ABB RAPID module: SetupWO.mod

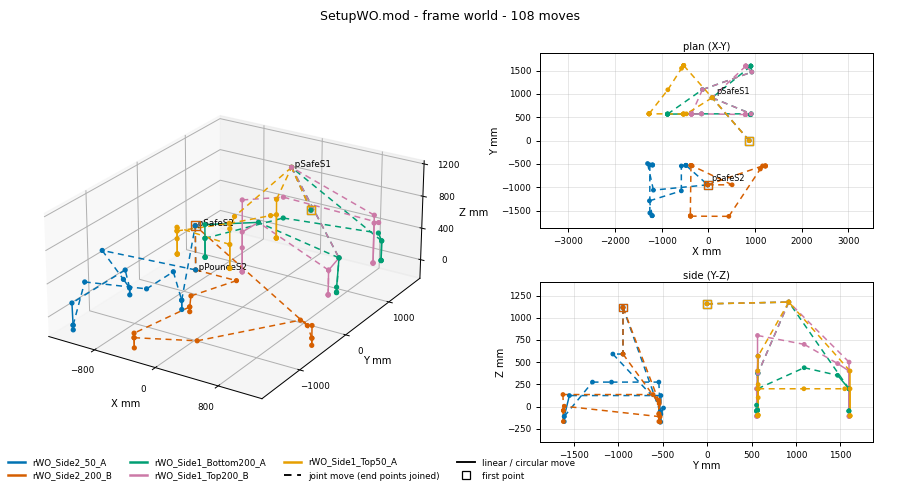
[picture p0: tool path of SetupWO.mod in frame world, 108 of 108 moves have a stored position in this frame; points joined in program order, loops and branches not executed]
MODULE SetupWO
	CONST robtarget pPounceS11:=[[-35.68,-1481.68,-160.88],[0.0139857,0.369962,0.928841,-0.0136566],[-2,1,-2,0],[9E+09,9E+09,9E+09,9E+09,9E+09,9E+09]];
	CONST robtarget pPounceS12:=[[1323.92,1454.10,-169.98],[0.00216079,-0.276188,0.961084,0.00568097],[0,-2,1,0],[9E+09,9E+09,9E+09,9E+09,9E+09,9E+09]];
	CONST robtarget pSafeS91:=[[-851.55,865.08,638.38],[0.0987927,0.977932,-0.183201,0.0180468],[1,0,-1,0],[9E+09,9E+09,9E+09,9E+09,9E+09,9E+09]];
	PROC rWO_Side2_50_A()
		MoveJ pSafeS2, v800, fine, tWeldGun;
		MoveJ pPounceS2, v800, fine, tWeldGun;
		MoveJ [[-1175.59,-1061.41,590.91],[0.0290518,0.998376,-0.0425584,0.0242723],[-2,-1,0,0],[9E+09,9E+09,9E+09,9E+09,9E+09,9E+09]], v800, z10, tWeldGun;
		MoveJ [[-1300.83,-491.42,-17.13],[0.0290285,0.998379,-0.0425044,0.0242811],[-2,-2,1,0],[9E+09,9E+09,9E+09,9E+09,9E+09,9E+09]], v800, z10, tWeldGun;
		MoveL [[-1195.07,-522.25,-85.28],[0.0287714,0.998373,-0.0426242,0.0246318],[-2,-2,1,0],[9E+09,9E+09,9E+09,9E+09,9E+09,9E+09]], v800, z10, tWeldGun;
		X1:
		MoveL [[-1195.09,-522.33,-173.98],[0.0287773,0.998376,-0.042547,0.0246393],[-2,-2,1,0],[9E+09,9E+09,9E+09,9E+09,9E+09,9E+09]], v800, fine, tWeldGun;
		MoveL [[-1195.07,-522.24,-85.28],[0.0287708,0.998373,-0.0426249,0.0246327],[-2,-2,1,0],[9E+09,9E+09,9E+09,9E+09,9E+09,9E+09]], v800, z10, tWeldGun;
		MoveJ [[-1253.08,-520.20,123.53],[0.0289856,0.998373,-0.0426291,0.0243837],[-2,-2,1,0],[9E+09,9E+09,9E+09,9E+09,9E+09,9E+09]], v800, z10, tWeldGun;
		MoveJ [[-1252.34,-1550.77,123.51],[0.0289915,0.998371,-0.0426611,0.0243853],[-2,-1,1,0],[9E+09,9E+09,9E+09,9E+09,9E+09,9E+09]], v800, z10, tWeldGun;
		MoveL [[-1203.52,-1608.74,-112.11],[0.0144898,0.998681,-0.0423691,0.0251074],[-2,-1,1,0],[9E+09,9E+09,9E+09,9E+09,9E+09,9E+09]], v800, z10, tWeldGun;
		X2:
		MoveL [[-1203.58,-1608.77,-169.27],[0.0144836,0.998684,-0.0423489,0.025044],[-2,-1,1,0],[9E+09,9E+09,9E+09,9E+09,9E+09,9E+09]], v800, fine, tWeldGun;
		MoveL [[-1203.52,-1608.74,-112.11],[0.0144918,0.998681,-0.0423701,0.0251105],[-2,-1,1,0],[9E+09,9E+09,9E+09,9E+09,9E+09,9E+09]], v800, z10, tWeldGun;
		MoveJ [[-1260.62,-1290.63,274.96],[0.0145241,0.998684,-0.0422942,0.0250997],[-2,-1,1,0],[9E+09,9E+09,9E+09,9E+09,9E+09,9E+09]], v800, z10, tWeldGun;
		MoveJ [[-577.42,-1076.50,274.99],[0.0145152,0.998684,-0.042322,0.0250813],[-2,-1,1,0],[9E+09,9E+09,9E+09,9E+09,9E+09,9E+09]], v800, z10, tWeldGun;
		MoveJ [[-577.39,-543.42,274.98],[0.0145354,0.998682,-0.0423423,0.0251146],[-2,-1,1,0],[9E+09,9E+09,9E+09,9E+09,9E+09,9E+09]], v800, z10, tWeldGun;
		MoveJ [[-478.99,-529.16,-59.08],[0.0144521,0.998675,-0.0425363,0.0251153],[-2,-2,1,0],[9E+09,9E+09,9E+09,9E+09,9E+09,9E+09]], v800, z10, tWeldGun;
		Y1:
		MoveL [[-479.00,-529.24,-174.87],[0.0144769,0.998677,-0.0424711,0.0251064],[-2,-2,2,0],[9E+09,9E+09,9E+09,9E+09,9E+09,9E+09]], v800, fine, tWeldGun;
		MoveL [[-478.99,-529.16,-59.08],[0.0144527,0.998675,-0.0425336,0.0251147],[-2,-2,1,0],[9E+09,9E+09,9E+09,9E+09,9E+09,9E+09]], v800, z10, tWeldGun;
		MoveJ pSafeS2, v800, fine, tWeldGun;
	ENDPROC
	PROC rWO_Side2_200_B()
		MoveJ pSafeS2, v800, fine, tWeldGun;
		MoveJ pPounceS2, v800, fine, tWeldGun;
		MoveJ [[510.39,-947.34,590.96],[0.00440116,-0.169072,0.985593,-0.00107979],[-1,0,-2,0],[9E+09,9E+09,9E+09,9E+09,9E+09,9E+09]], v800, z10, tWeldGun;
		MoveJ [[-346.53,-539.81,31.85],[0.00581128,-0.165183,0.98623,-0.00561328],[-2,0,-2,0],[9E+09,9E+09,9E+09,9E+09,9E+09,9E+09]], v800, z10, tWeldGun;
		MoveL [[-370.69,-531.16,-114.28],[0.00581574,-0.165115,0.986242,-0.00552901],[-2,0,-2,0],[9E+09,9E+09,9E+09,9E+09,9E+09,9E+09]], v800, z10, tWeldGun;
		X1:
		MoveL [[-370.69,-531.24,-173.68],[0.00581718,-0.165073,0.986249,-0.00556015],[-2,0,-2,0],[9E+09,9E+09,9E+09,9E+09,9E+09,9E+09]], v800, fine, tWeldGun;
		MoveL [[-370.69,-531.16,-114.28],[0.00581398,-0.165115,0.986242,-0.00552968],[-2,0,-2,0],[9E+09,9E+09,9E+09,9E+09,9E+09,9E+09]], v800, z10, tWeldGun;
		MoveJ [[-385.03,-1608.16,3.65],[0.0114791,0.162686,-0.986611,-0.000640749],[-2,0,-2,0],[9E+09,9E+09,9E+09,9E+09,9E+09,9E+09]], v800, z10, tWeldGun;
		MoveL [[-378.93,-1618.74,-45.41],[0.0114675,0.162653,-0.986616,-0.00066149],[-2,0,-2,0],[9E+09,9E+09,9E+09,9E+09,9E+09,9E+09]], v800, z10, tWeldGun;
		X2:
		MoveL [[-378.92,-1618.72,-168.89],[0.0114569,0.162671,-0.986614,-0.000676414],[-2,0,-2,0],[9E+09,9E+09,9E+09,9E+09,9E+09,9E+09]], v800, fine, tWeldGun;
		MoveL [[-378.94,-1618.74,-45.41],[0.0114698,0.162654,-0.986616,-0.000662067],[-2,0,-2,0],[9E+09,9E+09,9E+09,9E+09,9E+09,9E+09]], v800, z10, tWeldGun;
		MoveJ [[440.69,-1623.12,134.87],[0.0113911,0.162747,-0.986602,-0.000677745],[-1,0,-2,0],[9E+09,9E+09,9E+09,9E+09,9E+09,9E+09]], v800, z10, tWeldGun;
		MoveJ [[1115.37,-608.24,134.88],[0.0113576,0.162675,-0.986614,-0.000752857],[-1,0,-2,0],[9E+09,9E+09,9E+09,9E+09,9E+09,9E+09]], v800, z10, tWeldGun;
		MoveJ [[1224.24,-543.24,71.46],[0.0113815,0.162615,-0.986624,-0.000792876],[-1,0,-2,0],[9E+09,9E+09,9E+09,9E+09,9E+09,9E+09]], v800, z10, tWeldGun;
		MoveL [[1224.25,-543.16,-81.76],[0.0113472,0.162628,-0.986622,-0.000837926],[-1,1,-2,0],[9E+09,9E+09,9E+09,9E+09,9E+09,9E+09]], v800, z10, tWeldGun;
		Y1:
		MoveL [[1224.31,-543.22,-168.88],[0.0113297,0.162634,-0.986621,-0.000795503],[-1,1,-2,0],[9E+09,9E+09,9E+09,9E+09,9E+09,9E+09]], v800, fine, tWeldGun;
		MoveL [[1224.24,-543.16,-81.76],[0.0113488,0.162628,-0.986622,-0.000839478],[-1,1,-2,0],[9E+09,9E+09,9E+09,9E+09,9E+09,9E+09]], v800, z10, tWeldGun;
		MoveJ [[1164.77,-541.67,54.80],[0.0113578,0.162695,-0.986611,-0.000809552],[-1,0,-2,0],[9E+09,9E+09,9E+09,9E+09,9E+09,9E+09]], v800, z10, tWeldGun;
		MoveJ pSafeS2, v800, fine, tWeldGun;
	ENDPROC
	PROC rWO_Side1_Bottom200_A()
		MoveJ [[877.74,-1.13,1156.39],[0.00629862,0.00175411,0.999978,-0.000493005],[0,-1,0,0],[9E+09,9E+09,9E+09,9E+09,9E+09,9E+09]], v1000, z50, tWeldGun;
		TPWrite "200 Gallon Final S1 A setup wobj";
		MoveJ pSafeS1, v800, fine, tWeldGun;
		MoveJ [[918.61,573.57,375.55],[0.00167632,0.982899,-0.180568,0.0360764],[0,0,-2,0],[9E+09,9E+09,9E+09,9E+09,9E+09,9E+09]], v800, fine, tWeldGun;
		MoveL [[904.80,556.57,15.08],[0.00175291,0.982905,-0.180533,0.0360872],[0,0,-2,0],[9E+09,9E+09,9E+09,9E+09,9E+09,9E+09]], v800, fine, tWeldGun;
		MoveL [[904.79,556.65,-48.58],[0.00170966,0.982899,-0.180573,0.0360536],[0,0,-2,0],[9E+09,9E+09,9E+09,9E+09,9E+09,9E+09]], v800, fine, tWeldGun;
		x1:
		MoveL [[904.78,556.65,-53.58],[0.00170821,0.982899,-0.180576,0.0360527],[0,0,-2,0],[9E+09,9E+09,9E+09,9E+09,9E+09,9E+09]], v800, fine, tWeldGun;
		MoveL [[904.79,556.65,-48.58],[0.00170966,0.982899,-0.180573,0.0360536],[0,0,-2,0],[9E+09,9E+09,9E+09,9E+09,9E+09,9E+09]], v800, fine, tWeldGun;
		MoveJ [[918.61,573.57,375.55],[0.00167632,0.982899,-0.180568,0.0360764],[0,0,-2,0],[9E+09,9E+09,9E+09,9E+09,9E+09,9E+09]], v800, fine, tWeldGun;
		MoveJ [[-144.75,573.72,567.04],[0.00167262,0.982899,-0.180569,0.036075],[0,0,-2,0],[9E+09,9E+09,9E+09,9E+09,9E+09,9E+09]], v800, fine, tWeldGun;
		MoveL [[-872.91,567.93,374.12],[0.00165456,0.982899,-0.180556,0.036133],[1,0,-1,0],[9E+09,9E+09,9E+09,9E+09,9E+09,9E+09]], v800, fine, tWeldGun;
		MoveL [[-872.93,567.95,200],[0.00164969,0.982897,-0.180575,0.0361151],[1,1,-2,0],[9E+09,9E+09,9E+09,9E+09,9E+09,9E+09]], v800, fine, tWeldGun;
		MoveL [[-872.93,567.95,-39.59],[0.00164937,0.982897,-0.180575,0.0361144],[1,1,-2,0],[9E+09,9E+09,9E+09,9E+09,9E+09,9E+09]], v800, fine, tWeldGun;
		Y1:
		MoveL [[-872.93,567.95,-44.59],[0.00164864,0.982897,-0.180572,0.0361148],[1,1,-2,0],[9E+09,9E+09,9E+09,9E+09,9E+09,9E+09]], v800, fine, tWeldGun;
		MoveL [[-872.93,567.95,-39.59],[0.00164937,0.982897,-0.180575,0.0361144],[1,1,-2,0],[9E+09,9E+09,9E+09,9E+09,9E+09,9E+09]], v800, fine, tWeldGun;
		MoveL [[-872.93,567.95,200],[0.00164969,0.982897,-0.180575,0.0361151],[1,1,-2,0],[9E+09,9E+09,9E+09,9E+09,9E+09,9E+09]], v800, fine, tWeldGun;
		MoveJ [[-125.15,1093.11,436.96],[0.00164383,0.982897,-0.180567,0.0361424],[0,0,-2,0],[9E+09,9E+09,9E+09,9E+09,9E+09,9E+09]], v800, fine, tWeldGun;
		MoveJ [[933.14,1469.07,351.37],[0.00168757,0.982899,-0.180555,0.0361338],[0,0,-2,0],[9E+09,9E+09,9E+09,9E+09,9E+09,9E+09]], v800, fine, tWeldGun;
		MoveL [[911.23,1596.48,200],[0.00170312,0.982901,-0.180549,0.0361329],[0,0,-2,0],[9E+09,9E+09,9E+09,9E+09,9E+09,9E+09]], v800, fine, tWeldGun;
		MoveL [[911.23,1596.48,-48.8],[0.00170391,0.9829,-0.180551,0.0361313],[0,0,-2,0],[9E+09,9E+09,9E+09,9E+09,9E+09,9E+09]], v800, fine, tWeldGun;
		X2:
		MoveL [[911.23,1596.48,-53.80],[0.00170506,0.982901,-0.180548,0.0361311],[0,0,-2,0],[9E+09,9E+09,9E+09,9E+09,9E+09,9E+09]], v800, fine, tWeldGun;
		MoveL [[911.23,1596.48,-48.81],[0.00170363,0.982901,-0.18055,0.0361308],[0,0,-2,0],[9E+09,9E+09,9E+09,9E+09,9E+09,9E+09]], v800, fine, tWeldGun;
		MoveL [[911.23,1596.48,200],[0.00170784,0.982901,-0.180549,0.0361301],[0,0,-2,0],[9E+09,9E+09,9E+09,9E+09,9E+09,9E+09]], v800, fine, tWeldGun;
		MoveJ pSafeS1, v800, fine, tWeldGun;
	ENDPROC
	PROC rWO_Side1_Top200_B()
		MoveJ [[877.74,-1.13,1156.39],[0.00629862,0.00175411,0.999978,-0.000493005],[0,-1,0,0],[9E+09,9E+09,9E+09,9E+09,9E+09,9E+09]], v1000, z50, tWeldGun;
		MoveJ pSafeS1, v800, fine, tWeldGun;
		MoveJ [[918.61,573.57,375.55],[0.00167632,0.982899,-0.180568,0.0360764],[0,0,-2,0],[9E+09,9E+09,9E+09,9E+09,9E+09,9E+09]], v800, fine, tWeldGun;
		MoveL [[795.8,558.19,200],[0.00172974,0.9829,-0.18057,0.0360319],[0,0,-2,0],[9E+09,9E+09,9E+09,9E+09,9E+09,9E+09]], v800, fine, tWeldGun;
		MoveL [[795.8,558.19,-106.62],[0.00173069,0.982901,-0.180568,0.0360302],[0,0,-2,0],[9E+09,9E+09,9E+09,9E+09,9E+09,9E+09]], v800, fine, tWeldGun;
		x1:
		MoveL [[795.80,558.18,-111.62],[0.00173128,0.982901,-0.180567,0.0360306],[0,0,-2,0],[9E+09,9E+09,9E+09,9E+09,9E+09,9E+09]], v800, fine, tWeldGun;
		MoveL [[795.8,558.18,-106.62],[0.00173073,0.982901,-0.180569,0.0360303],[0,0,-2,0],[9E+09,9E+09,9E+09,9E+09,9E+09,9E+09]], v800, fine, tWeldGun;
		MoveJ [[795.8,558.19,200],[0.00172993,0.9829,-0.180571,0.0360296],[0,0,-2,0],[9E+09,9E+09,9E+09,9E+09,9E+09,9E+09]], v800, fine, tWeldGun;
		MoveJ [[-144.75,573.72,567.04],[0.00167262,0.982899,-0.180569,0.036075],[0,0,-2,0],[9E+09,9E+09,9E+09,9E+09,9E+09,9E+09]], v800, fine, tWeldGun;
		MoveJ [[-144.74,573.74,567.05],[0.0333231,-0.167825,0.985155,-0.0139539],[1,-1,1,0],[9E+09,9E+09,9E+09,9E+09,9E+09,9E+09]], v800, fine, tWeldGun;
		MoveL [[-360.28,567.56,400],[0.0326173,-0.214911,0.975965,-0.0155425],[1,-1,1,0],[9E+09,9E+09,9E+09,9E+09,9E+09,9E+09]], v800, fine, tWeldGun;
		MoveL [[-360.28,567.57,200],[0.0326196,-0.214908,0.975966,-0.0155416],[1,-1,1,0],[9E+09,9E+09,9E+09,9E+09,9E+09,9E+09]], v800, fine, tWeldGun;
		MoveL [[-360.28,567.56,-103.19],[0.0326171,-0.21491,0.975965,-0.0155414],[1,-1,1,0],[9E+09,9E+09,9E+09,9E+09,9E+09,9E+09]], v800, fine, tWeldGun;
		Y1:
		MoveL [[-360.28,567.56,-108.19],[0.032618,-0.21491,0.975965,-0.0155432],[1,-1,1,0],[9E+09,9E+09,9E+09,9E+09,9E+09,9E+09]], v800, fine, tWeldGun;
		MoveL [[-360.28,567.56,-103.19],[0.0326174,-0.214911,0.975965,-0.0155431],[1,-1,1,0],[9E+09,9E+09,9E+09,9E+09,9E+09,9E+09]], v800, fine, tWeldGun;
		MoveL [[-360.28,567.57,800],[0.0326175,-0.214911,0.975965,-0.0155423],[1,-1,1,0],[9E+09,9E+09,9E+09,9E+09,9E+09,9E+09]], v800, fine, tWeldGun;
		MoveJ [[-125.15,1093.11,700],[0.00164383,0.982897,-0.180567,0.0361424],[0,0,-2,0],[9E+09,9E+09,9E+09,9E+09,9E+09,9E+09]], v800, fine, tWeldGun;
		MoveJ [[933.13,1469.10,483.55],[0.00167665,0.982898,-0.180566,0.0361131],[0,0,-2,0],[9E+09,9E+09,9E+09,9E+09,9E+09,9E+09]], v800, fine, tWeldGun;
		MoveL [[804.15,1598.36,400],[0.00171595,0.982897,-0.180572,0.0361275],[0,0,-2,0],[9E+09,9E+09,9E+09,9E+09,9E+09,9E+09]], v800, fine, tWeldGun;
		MoveL [[804.15,1598.36,-108.05],[0.00171494,0.982897,-0.180572,0.0361272],[0,0,-2,0],[9E+09,9E+09,9E+09,9E+09,9E+09,9E+09]], v800, fine, tWeldGun;
		X2:
		MoveL [[804.15,1598.36,-113.05],[0.00171524,0.982897,-0.180571,0.0361286],[0,0,-2,0],[9E+09,9E+09,9E+09,9E+09,9E+09,9E+09]], v800, fine, tWeldGun;
		MoveL [[804.16,1598.36,-108.05],[0.001714,0.982896,-0.180572,0.0361276],[0,0,-2,0],[9E+09,9E+09,9E+09,9E+09,9E+09,9E+09]], v800, fine, tWeldGun;
		MoveL [[804.15,1598.36,500],[0.00171494,0.982897,-0.180571,0.036128],[0,0,-2,0],[9E+09,9E+09,9E+09,9E+09,9E+09,9E+09]], v800, fine, tWeldGun;
		MoveJ pSafeS1, v800, fine, tWeldGun;
	ENDPROC
	PROC rWO_Side1_Top50_A()
		MoveJ [[877.74,-1.13,1156.39],[0.00629862,0.00175411,0.999978,-0.000493005],[0,-1,0,0],[9E+09,9E+09,9E+09,9E+09,9E+09,9E+09]], v1000, z50, tWeldGun;
		MoveJ pSafeS1, v800, fine, tWeldGun;
		MoveJ [[-468.95,573.70,567.01],[0.0333012,-0.16781,0.985157,-0.0139911],[1,-1,1,0],[9E+09,9E+09,9E+09,9E+09,9E+09,9E+09]], v800, fine, tWeldGun;
		MoveL [[-531.39,570.33,400],[0.0326975,-0.214889,0.975966,-0.0155984],[1,-1,1,0],[9E+09,9E+09,9E+09,9E+09,9E+09,9E+09]], v800, fine, tWeldGun;
		MoveL [[-532.73,569.16,-101.03],[0.0149429,0.21368,-0.976372,0.0285468],[1,-1,1,0],[9E+09,9E+09,9E+09,9E+09,9E+09,9E+09]], v800, fine, tWeldGun;
		x1:
		MoveL [[-532.72,569.15,-106.04],[0.0149421,0.213677,-0.976373,0.0285481],[1,-1,1,0],[9E+09,9E+09,9E+09,9E+09,9E+09,9E+09]], v800, fine, tWeldGun;
		MoveL [[-532.73,569.16,-101.03],[0.0149438,0.213678,-0.976373,0.0285467],[1,-1,1,0],[9E+09,9E+09,9E+09,9E+09,9E+09,9E+09]], v800, fine, tWeldGun;
		MoveL [[-531.38,570.32,200],[0.0327034,-0.214883,0.975967,-0.0156014],[1,-1,1,0],[9E+09,9E+09,9E+09,9E+09,9E+09,9E+09]], v800, fine, tWeldGun;
		MoveJ [[-1268.46,574.85,247.14],[0.032725,-0.214887,0.975966,-0.0155941],[1,-1,1,0],[9E+09,9E+09,9E+09,9E+09,9E+09,9E+09]], v800, fine, tWeldGun;
		MoveL [[-1268.46,574.83,200],[0.0327132,-0.21488,0.975968,-0.0156117],[1,-1,1,0],[9E+09,9E+09,9E+09,9E+09,9E+09,9E+09]], v800, fine, tWeldGun;
		MoveL [[-1268.45,574.83,100],[0.0327149,-0.214878,0.975968,-0.0156121],[1,-1,1,0],[9E+09,9E+09,9E+09,9E+09,9E+09,9E+09]], v800, fine, tWeldGun;
		MoveL [[-1269.03,574.3,-95.71],[0.00752882,-0.214386,0.976491,-0.0211491],[1,-1,1,0],[9E+09,9E+09,9E+09,9E+09,9E+09,9E+09]], v800, fine, tWeldGun;
		Y1:
		MoveL [[-1269.03,574.30,-100.71],[0.00752894,-0.214385,0.976491,-0.0211483],[1,-1,1,0],[9E+09,9E+09,9E+09,9E+09,9E+09,9E+09]], v800, fine, tWeldGun;
		MoveL [[-1269.03,574.3,-95.71],[0.00752919,-0.214386,0.976491,-0.0211493],[1,-1,1,0],[9E+09,9E+09,9E+09,9E+09,9E+09,9E+09]], v800, fine, tWeldGun;
		MoveL [[-1268.46,574.83,200],[0.0327153,-0.214879,0.975968,-0.0156123],[1,-1,1,0],[9E+09,9E+09,9E+09,9E+09,9E+09,9E+09]], v800, fine, tWeldGun;
		MoveJ [[-866.78,1089.37,199.98],[0.0327388,-0.214897,0.975963,-0.0155931],[1,-1,1,0],[9E+09,9E+09,9E+09,9E+09,9E+09,9E+09]], v800, fine, tWeldGun;
		MoveJ [[-573.13,1549.48,199.96],[0.0327434,-0.214866,0.975971,-0.0155433],[1,-1,1,0],[9E+09,9E+09,9E+09,9E+09,9E+09,9E+09]], v800, fine, tWeldGun;
		MoveL [[-527.05,1609.12,200],[0.0294376,0.214786,-0.97608,0.0163697],[1,-1,1,0],[9E+09,9E+09,9E+09,9E+09,9E+09,9E+09]], v800, fine, tWeldGun;
		MoveL [[-527.06,1609.11,-102.87],[0.0294363,0.214784,-0.976081,0.01637],[1,-1,1,0],[9E+09,9E+09,9E+09,9E+09,9E+09,9E+09]], v800, fine, tWeldGun;
		X2:
		MoveL [[-527.06,1609.11,-107.87],[0.0294376,0.214784,-0.97608,0.0163707],[1,-1,1,0],[9E+09,9E+09,9E+09,9E+09,9E+09,9E+09]], v800, fine, tWeldGun;
		MoveL [[-527.05,1609.11,-102.87],[0.0294374,0.214783,-0.976081,0.0163714],[1,-1,1,0],[9E+09,9E+09,9E+09,9E+09,9E+09,9E+09]], v800, fine, tWeldGun;
		MoveL [[-527.05,1609.11,400],[0.0294374,0.214786,-0.97608,0.0163704],[1,-1,1,0],[9E+09,9E+09,9E+09,9E+09,9E+09,9E+09]], v800, fine, tWeldGun;
		MoveJ pSafeS1, v800, fine, tWeldGun;
	ENDPROC

ENDMODULE
